// Mitsubishi GX Works2 project: PLC_Group14   PLC: FX3G

// global labels: Global1
VAR_GLOBAL
  StartDay AT X007 : BOOL;
  Start_day AT X007 : BOOL;
  Start_indicator AT Y007 : BOOL;
  emg_buttom AT X005 : BOOL;
  Storage_indicator AT M5 : BOOL;
  Storage_Check AT X010 : BOOL;
  minimum_chocolate AT K400 : INT;
  Chocolate_Min AT M1 : BOOL;
  Nuts_Storage AT D1603 : REAL;
  minimun_nuts AT K100 : INT;
  Nuts_Min AT M2 : BOOL;
  Fistuk_Storage AT D1703 : REAL;
  minumum_fistuk AT K120 : INT;
  fistuk : BOOL;
  Fistuk_Min AT M3 : BOOL;
  Kadaif_Storage AT D1803 : REAL;
  minimum_kadaif AT K60 : INT;
  Kadaif_Min AT M4 : BOOL;
  input_storage AT X007 : BOOL;
  initial_chocolate AT D1500 : REAL;
  initial_nuts AT D1600 : REAL;
  initial_fistuk AT D1700 : REAL;
  initial_kadaif AT D1800 : REAL;
  Chocolate_Storage AT D1503 : REAL;
  Ch_amount AT E400 : REAL;
  melt_time AT TC1 : BOOL;
END_VAR
VAR_GLOBAL CONSTANT
  five40 : INT := 40;
  four_sec : INT := 40;
END_VAR
VAR_GLOBAL
  melt_indictor AT Y001 : BOOL;
  timer_melt_finish AT TS1 : BOOL;
  location_time AT TC2 : BOOL;
END_VAR
VAR_GLOBAL CONSTANT
  two_sec : INT := 20;
END_VAR
VAR_GLOBAL
  location_time_finish AT TS2 : BOOL;
  pouring_time AT TC3 : BOOL;
  pouring_time_finish AT TS3 : BOOL;
  pouring_indictor AT Y002 : BOOL;
END_VAR
VAR_GLOBAL CONSTANT
  six_sec : INT := 60;
END_VAR
VAR_GLOBAL
  input_buttom AT X004 : BOOL;
  analog_input_1 AT D8280 : INT;
END_VAR
VAR_GLOBAL CONSTANT
  Normalizer : INT := 400;
END_VAR
VAR_GLOBAL
  ch_type AT D1900 : REAL;
END_VAR
VAR_GLOBAL CONSTANT
  ch_mix_nuts : REAL := 4;
  ch_dubai : REAL := 4;
END_VAR
VAR_GLOBAL
  dubai_light AT M7 : BOOL;
  mix_nuts_light AT M6 : BOOL;
END_VAR
VAR_GLOBAL CONSTANT
  ch_mix : REAL := 5;
END_VAR
VAR_GLOBAL
  mix_nuts_for_sure AT M8 : BOOL;
  Nuts_Amount AT E20 : REAL;
  Fistuk_Amount AT E120 : REAL;
  Kadaif_Amount AT E60 : REAL;
  Nuts_Amount_mix AT E100 : REAL;
  Fistuk_Amount_mix AT E100 : REAL;
END_VAR
VAR_GLOBAL CONSTANT
  five_sec : INT := 50;
END_VAR
VAR_GLOBAL
  fill_creame_time AT TC4 : BOOL;
  timer_cream_finish AT TS4 : BOOL;
  fill_cream_time AT TC4 : BOOL;
  cream_indictor AT M9 : BOOL;
  help1 AT M10 : BOOL;
  light1 AT TC5 : BOOL;
END_VAR
VAR_GLOBAL CONSTANT
  half_sec : INT := 5;
END_VAR
VAR_GLOBAL
  light1_finish AT TS5 : BOOL;
  lamp_1 AT Y004 : BOOL;
  light2 AT TC6 : BOOL;
  light2_finish AT TS6 : BOOL;
  lamp_2 AT Y003 : BOOL;
  fliker_light AT M10 : BOOL;
  Cool_pros AT X006 : BOOL;
  Cool_time AT TC7 : BOOL;
END_VAR
VAR_GLOBAL CONSTANT
  three_sec : INT := 30;
END_VAR
VAR_GLOBAL
  Cool_time_finish AT TS7 : BOOL;
  Cool_light AT Y006 : BOOL;
  packing_pros AT X006 : BOOL;
  Counter_ch AT CC1 : BOOL;
  packing_buttom AT X000 : BOOL;
END_VAR
VAR_GLOBAL CONSTANT
  four_pack : INT := K4;
END_VAR
VAR_GLOBAL
  Cs AT M1 : BOOL;
  Cs_pack AT CS1 : BOOL;
  Packing_light AT Y005 : BOOL;
END_VAR
VAR_GLOBAL CONSTANT
  CON_1 : INT := K1;
END_VAR
VAR_GLOBAL
  Counter_ch_pack AT D2000 : REAL;
  analog_output AT D8282 : INT;
  Counter_ch_output AT D2100 : INT;
  temperture_indicator AT X002 : BOOL;
  location_indicator AT X003 : BOOL;
  end_day AT X010 : BOOL;
END_VAR
VAR_GLOBAL CONSTANT
  Normalizer1 : INT := 40;
END_VAR
VAR_GLOBAL
  end_d AT M13 : BOOL;
  melt_buttom AT X001 : BOOL;
END_VAR

// task Task_01 (event TRUE, interval 0, priority 31): POU_01

PROGRAM POU_01
(* structured ladder/FBD written out as ST: instructions are called as NAME(EN, inputs, outputs); _pN, _eN, _tN stand for wires *)
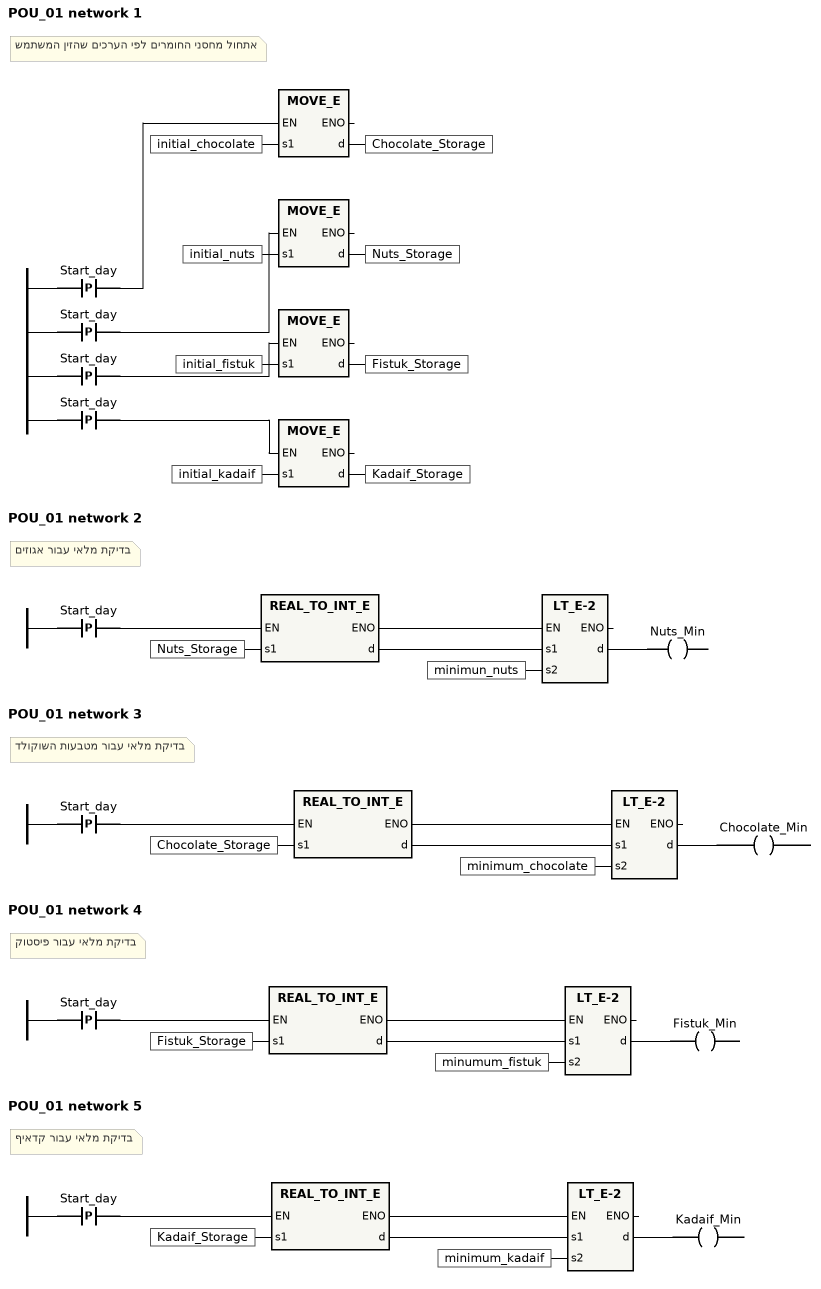
(* network 1 *)
(* אתחול מחסני החומרים לפי הערכים שהזין המשתמש *)
MOVE_E(LDP(TRUE, Start_day), initial_chocolate, Chocolate_Storage);
MOVE_E(LDP(TRUE, Start_day), initial_nuts, Nuts_Storage);
MOVE_E(LDP(TRUE, Start_day), initial_fistuk, Fistuk_Storage);
MOVE_E(LDP(TRUE, Start_day), initial_kadaif, Kadaif_Storage);
(* network 2 *)
(* בדיקת מלאי עבור אגוזים *)
_e2 := REAL_TO_INT_E(LDP(TRUE, Start_day), Nuts_Storage, _t1);
LT_E(_e2, _t1, minimun_nuts, _t3);
Nuts_Min := _t3;
(* network 3 *)
(* בדיקת מלאי עבור מטבעות השוקולד *)
_e2 := REAL_TO_INT_E(LDP(TRUE, Start_day), Chocolate_Storage, _t1);
LT_E(_e2, _t1, minimum_chocolate, _t3);
Chocolate_Min := _t3;
(* network 4 *)
(* בדיקת מלאי עבור פיסטוק *)
_e2 := REAL_TO_INT_E(LDP(TRUE, Start_day), Fistuk_Storage, _t1);
LT_E(_e2, _t1, minumum_fistuk, _t3);
Fistuk_Min := _t3;
(* network 5 *)
(* בדיקת מלאי עבור קדאיף *)
_e2 := REAL_TO_INT_E(LDP(TRUE, Start_day), Kadaif_Storage, _t1);
LT_E(_e2, _t1, minimum_kadaif, _t3);
Kadaif_Min := _t3;
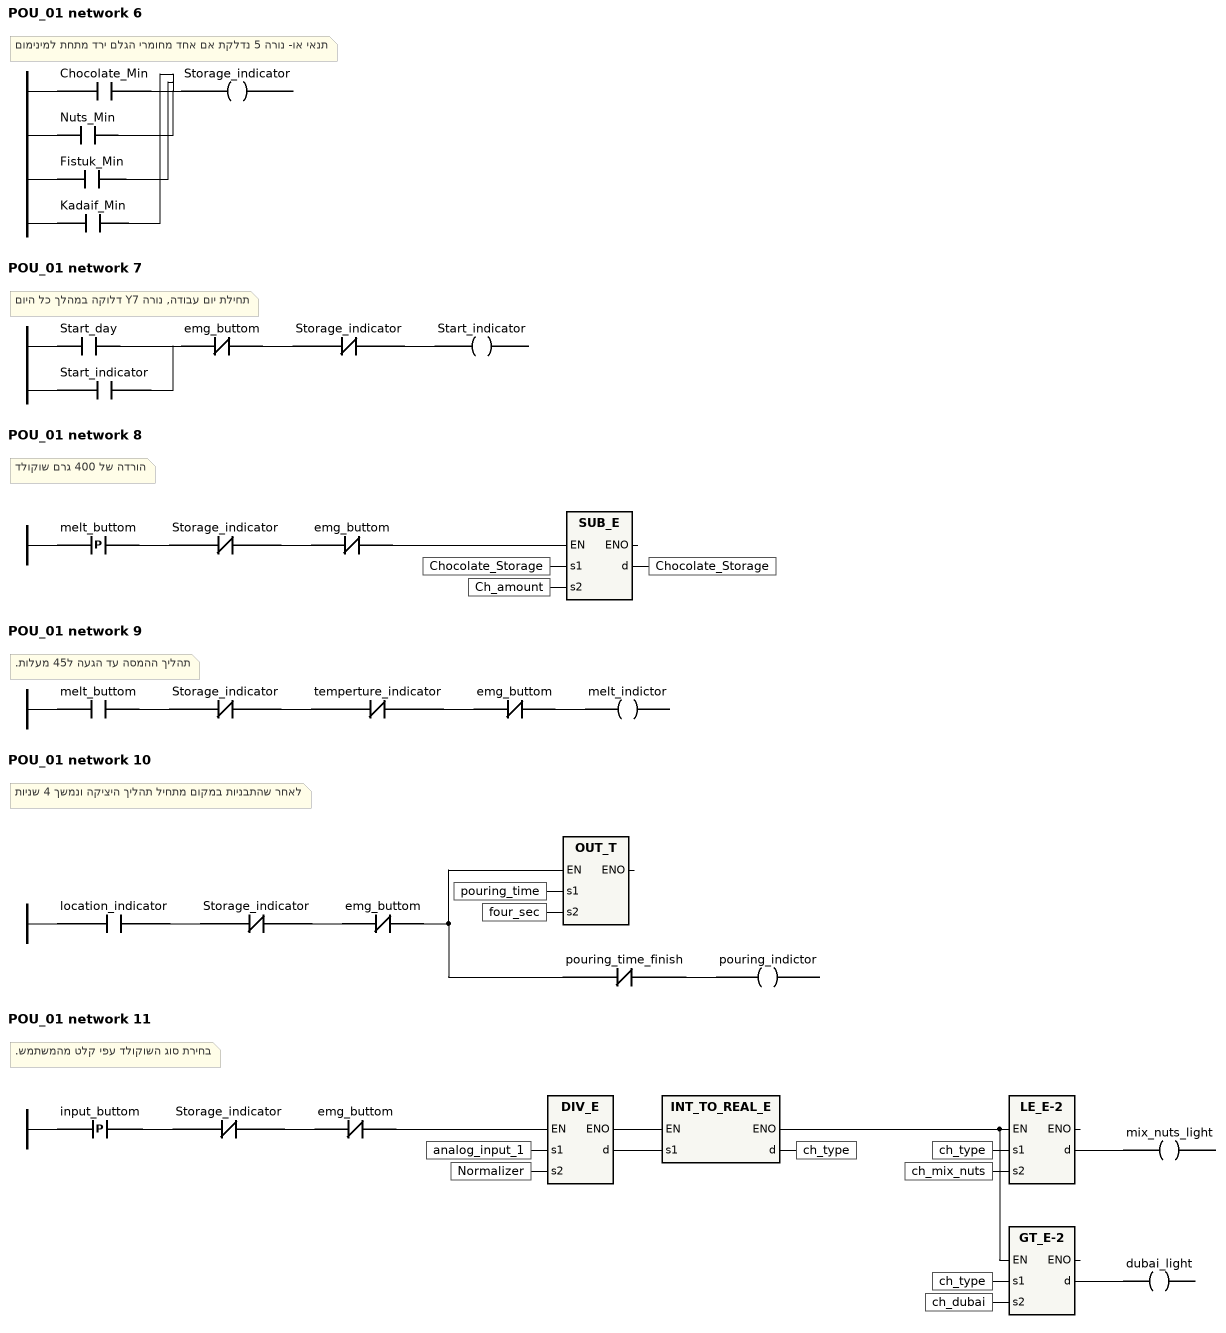
(* network 6 *)
(* תנאי או- נורה 5 נדלקת אם אחד מחומרי הגלם ירד מתחת למינימום *)
Storage_indicator := Chocolate_Min OR Nuts_Min OR Fistuk_Min OR Kadaif_Min;
(* network 7 *)
(* תחילת יום עבודה, נורה Y7 דלוקה במהלך כל היום *)
Start_indicator := ((Start_day OR Start_indicator) AND NOT emg_buttom) AND NOT Storage_indicator;
(* network 8 *)
(* הורדה של 400 גרם שוקולד *)
SUB_E(LDP(TRUE, melt_buttom) AND NOT Storage_indicator AND NOT emg_buttom, Chocolate_Storage, Ch_amount, Chocolate_Storage);
(* network 9 *)
(* תהליך ההמסה עד הגעה ל45 מעלות. *)
melt_indictor := melt_buttom AND NOT Storage_indicator AND NOT temperture_indicator AND NOT emg_buttom;
(* network 10 *)
(* לאחר שהתבניות במקום מתחיל תהליך היציקה ונמשך 4 שניות *)
_p1 := location_indicator AND NOT Storage_indicator AND NOT emg_buttom;
OUT_T(_p1, pouring_time, four_sec);
pouring_indictor := _p1 AND NOT pouring_time_finish;
(* network 11 *)
(* בחירת סוג השוקולד עפי קלט מהמשתמש. *)
_e2 := DIV_E(LDP(TRUE, input_buttom) AND NOT Storage_indicator AND NOT emg_buttom, analog_input_1, Normalizer, _t1);
_e3 := INT_TO_REAL_E(_e2, _t1, ch_type);
LE_E(_e3, ch_type, ch_mix_nuts, _t4);
mix_nuts_light := _t4;
GT_E(_e3, ch_type, ch_dubai, _t5);
dubai_light := _t5;
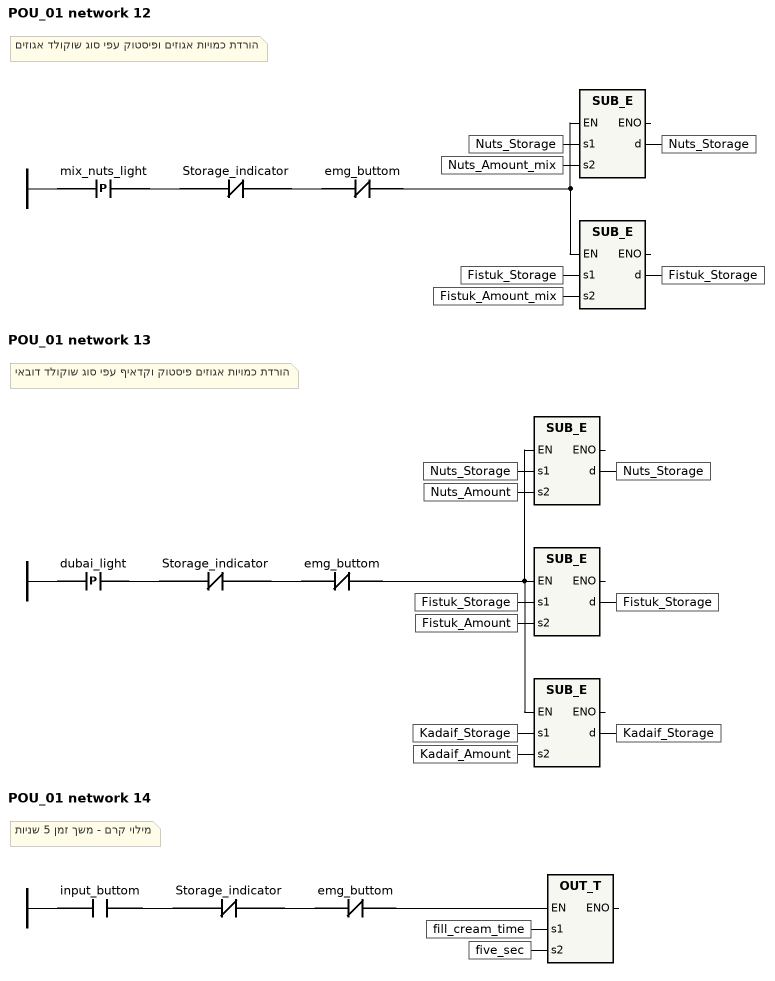
(* network 12 *)
(* הורדת כמויות אגוזים ופיסטוק עפי סוג שוקולד אגוזים *)
_p1 := LDP(TRUE, mix_nuts_light) AND NOT Storage_indicator AND NOT emg_buttom;
SUB_E(_p1, Nuts_Storage, Nuts_Amount_mix, Nuts_Storage);
SUB_E(_p1, Fistuk_Storage, Fistuk_Amount_mix, Fistuk_Storage);
(* network 13 *)
(* הורדת כמויות אגוזים פיסטוק וקדאיף עפי סוג שוקולד דובאי *)
_p1 := LDP(TRUE, dubai_light) AND NOT Storage_indicator AND NOT emg_buttom;
SUB_E(_p1, Nuts_Storage, Nuts_Amount, Nuts_Storage);
SUB_E(_p1, Fistuk_Storage, Fistuk_Amount, Fistuk_Storage);
SUB_E(_p1, Kadaif_Storage, Kadaif_Amount, Kadaif_Storage);
(* network 14 *)
(* מילוי קרם - משך זמן 5 שניות *)
OUT_T(input_buttom AND NOT Storage_indicator AND NOT emg_buttom, fill_cream_time, five_sec);
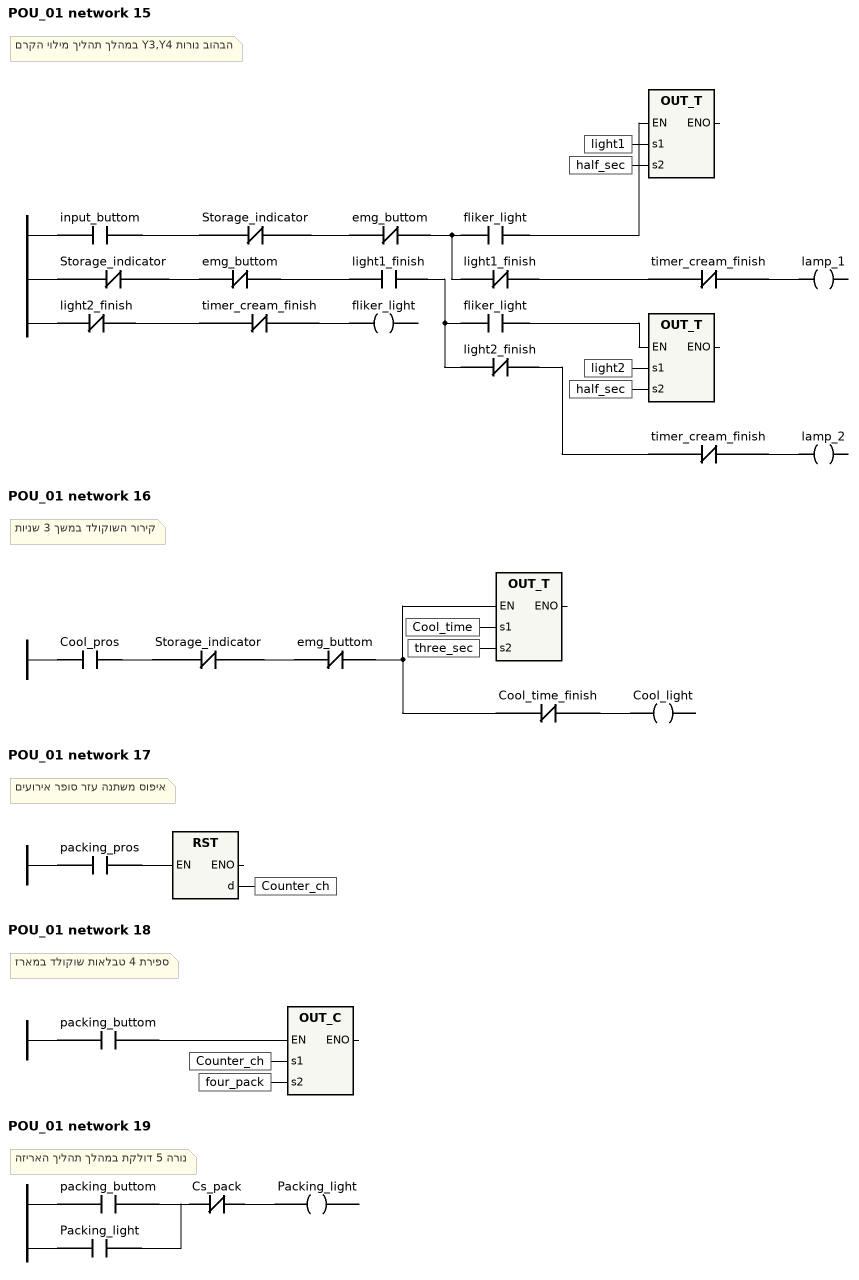
(* network 15 *)
(* הבהוב נורות Y3,Y4 במהלך תהליך מילוי הקרם *)
_p1 := input_buttom AND NOT Storage_indicator AND NOT emg_buttom;
OUT_T(_p1 AND fliker_light, light1, half_sec);
lamp_1 := _p1 AND NOT light1_finish AND NOT timer_cream_finish;
_p2 := NOT Storage_indicator AND NOT emg_buttom AND light1_finish;
OUT_T(_p2 AND fliker_light, light2, half_sec);
lamp_2 := _p2 AND NOT light2_finish AND NOT timer_cream_finish;
fliker_light := NOT light2_finish AND NOT timer_cream_finish;
(* network 16 *)
(* קירור השוקולד במשך 3 שניות *)
_p1 := Cool_pros AND NOT Storage_indicator AND NOT emg_buttom;
OUT_T(_p1, Cool_time, three_sec);
Cool_light := _p1 AND NOT Cool_time_finish;
(* network 17 *)
(* איפוס משתנה עזר סופר אירועים *)
RST(packing_pros, Counter_ch);
(* network 18 *)
(* ספירת 4 טבלאות שוקולד במארז *)
OUT_C(packing_buttom, Counter_ch, four_pack);
(* network 19 *)
(* נורה 5 דולקת במהלך תהליך האריזה *)
Packing_light := (packing_buttom OR Packing_light) AND NOT Cs_pack;
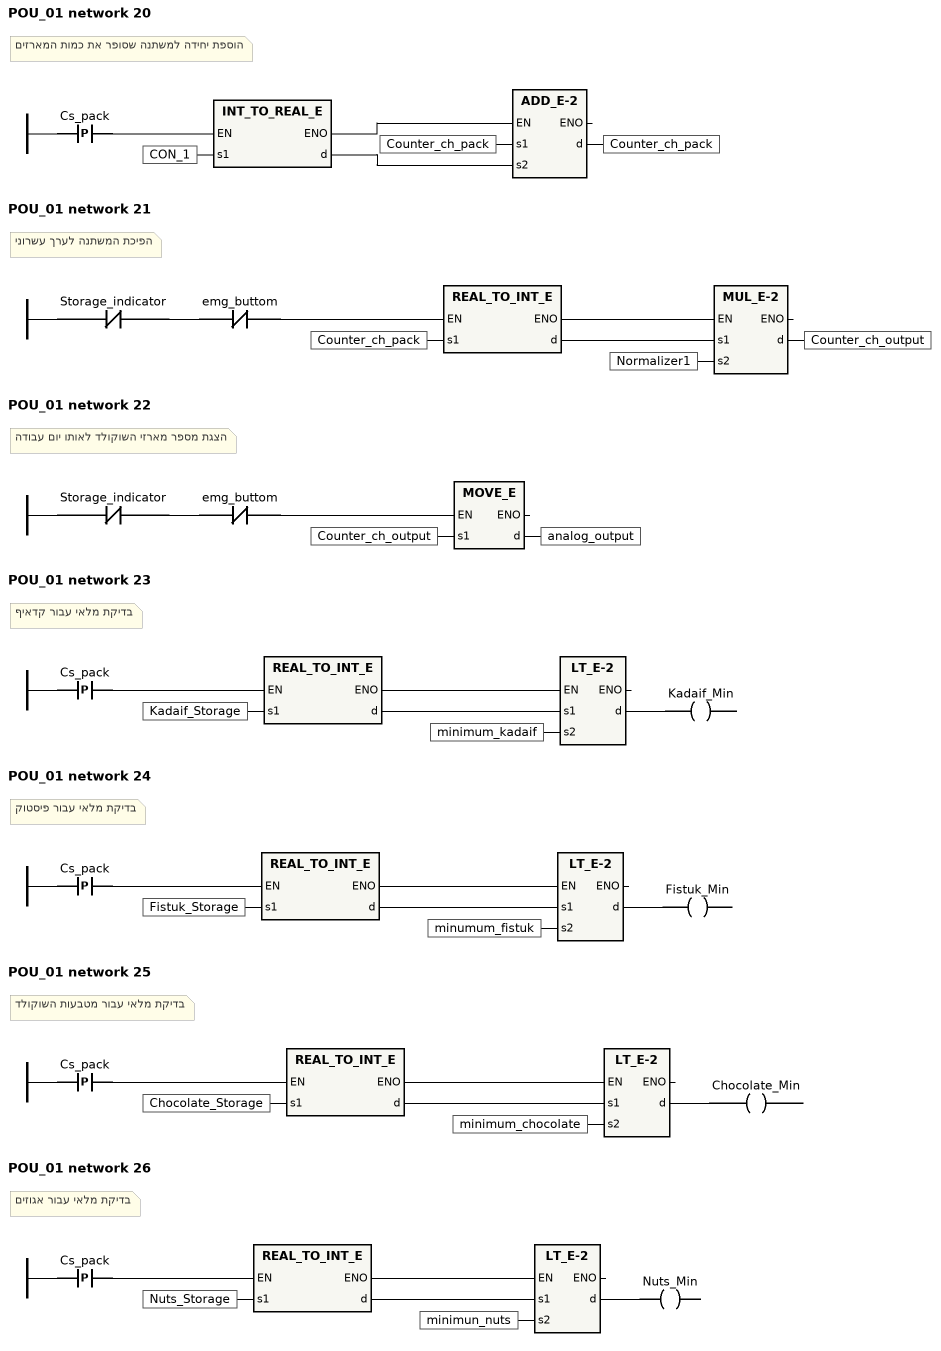
(* network 20 *)
(* הוספת יחידה למשתנה שסופר את כמות המארזים *)
_e2 := INT_TO_REAL_E(LDP(TRUE, Cs_pack), CON_1, _t1);
ADD_E(_e2, Counter_ch_pack, _t1, Counter_ch_pack);
(* network 21 *)
(* הפיכת המשתנה לערך עשרוני *)
_e2 := REAL_TO_INT_E(NOT Storage_indicator AND NOT emg_buttom, Counter_ch_pack, _t1);
MUL_E(_e2, _t1, Normalizer1, Counter_ch_output);
(* network 22 *)
(* הצגת מספר מארזי השוקולד לאותו יום עבודה *)
MOVE_E(NOT Storage_indicator AND NOT emg_buttom, Counter_ch_output, analog_output);
(* network 23 *)
(* בדיקת מלאי עבור קדאיף *)
_e2 := REAL_TO_INT_E(LDP(TRUE, Cs_pack), Kadaif_Storage, _t1);
LT_E(_e2, _t1, minimum_kadaif, _t3);
Kadaif_Min := _t3;
(* network 24 *)
(* בדיקת מלאי עבור פיסטוק *)
_e2 := REAL_TO_INT_E(LDP(TRUE, Cs_pack), Fistuk_Storage, _t1);
LT_E(_e2, _t1, minumum_fistuk, _t3);
Fistuk_Min := _t3;
(* network 25 *)
(* בדיקת מלאי עבור מטבעות השוקולד *)
_e2 := REAL_TO_INT_E(LDP(TRUE, Cs_pack), Chocolate_Storage, _t1);
LT_E(_e2, _t1, minimum_chocolate, _t3);
Chocolate_Min := _t3;
(* network 26 *)
(* בדיקת מלאי עבור אגוזים *)
_e2 := REAL_TO_INT_E(LDP(TRUE, Cs_pack), Nuts_Storage, _t1);
LT_E(_e2, _t1, minimun_nuts, _t3);
Nuts_Min := _t3;
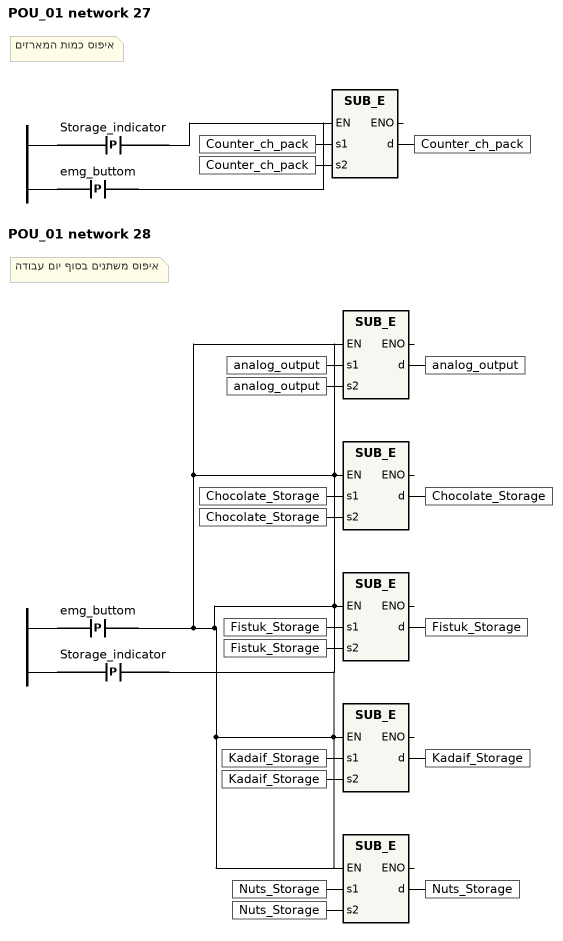
(* network 27 *)
(* איפוס כמות המארזים *)
SUB_E(LDP(TRUE, Storage_indicator) OR LDP(TRUE, emg_buttom), Counter_ch_pack, Counter_ch_pack, Counter_ch_pack);
(* network 28 *)
(* איפוס משתנים בסוף יום עבודה *)
_p1 := LDP(TRUE, emg_buttom) OR LDP(TRUE, Storage_indicator);
SUB_E(_p1, analog_output, analog_output, analog_output);
SUB_E(_p1, Chocolate_Storage, Chocolate_Storage, Chocolate_Storage);
SUB_E(_p1, Fistuk_Storage, Fistuk_Storage, Fistuk_Storage);
SUB_E(_p1, Kadaif_Storage, Kadaif_Storage, Kadaif_Storage);
SUB_E(_p1, Nuts_Storage, Nuts_Storage, Nuts_Storage);
END_PROGRAM
